(* CoDeSys 2.3.9.48 project: 5-hospital_Main_PLC.pro *)
(* Libraries: Standard.lib 20.5.14 09:13:26, Iecsfc.lib 30.1.13 14:05:12, SYSLIBCALLBACK.LIB 30.1.13 14:05:12, Modb_l05.lib 13.5.15 11:30:08, mod_com.lib 30.1.13 14:05:12, Serial_Interface_01.lib 22.4.13 13:50:14, SerComm.lib 30.1.13 14:05:12, Wago_MBCFG_SERIAL_01.lib 1.4.15 15:24:28, Wago_MBCFG_COMMON_01.lib 1.4.15 15:24:28 *)

(* PLC configuration (modules and I/O channels)
K-Bus [K_Bus] node 0, in %IB0 out %QB0 {KbusBusMode = 1; KbusCycleTime = 10000; KbusThreadPriority = 0; KbusSetOutputsToZeroOnApplicationStop = 1}
Modbus variables [PFC200MODBUS] node 1, in %IB0 out %QB0 {PlcStopBehaviour = 1; FiledbusErrorBehaviour = 1; TcpOperation = 1; TcpPort = 502; TcpTimeout = 600; UdpOperation = 1; UdpPort = 502; RtuOperation = 0; NodeId = 1; ResponseTimeout = 5000; Interface = 0; Baud = 115200; StopBits = 1; Parity = 1; FlowCtrl = 0; PhysInterface = 0}
Modbus-Master [MB_MASTER] node 2, in %IB0 out %QB0
*)

(* POU PLC_PRG, ST *)
PROGRAM PLC_PRG
VAR
END_VAR

END_PROGRAM

(* POU Generated Code/Serial/MBCFG/MBCFG_COM_OBJECTS, ST *)
PROGRAM MBCFG_COM_OBJECTS
VAR_INPUT

      MBCFG_MB_COM_0	:	MBCFG_COM_SER_OBJECT := (   ASCII_Mode      := FALSE,
                                                     COM_PORT        := 0,	 
                                                     COM_BAUDRATE    := BAUD_9600,
                                                     COM_PARITY      := PARITY_NO,
                                                     COM_STOPBITS    := STOPBITS_1,
                                                     COM_BYTESIZE    := BS_8,
                                                     COM_FLOW_CONTROL:= HALFDUPLEX,
                                                     TIME_OUT        := t#100ms
                                                 );



END_VAR
;
END_PROGRAM

(* POU Generated Code/Serial/MBCFG_ModbusSlave, ST *)
PROGRAM MBCFG_ModbusSlave (* generated by config one prg for each slave *)

VAR_INPUT

END_VAR

VAR_OUTPUT
           xNewVar       :    BOOL;       (**) 


    (*--- system variables (read only) -------------------------*)
    MBCFG_SlaveAddress  :   USINT := 1; (* valid range 1..247   *)
    MBCFG_TimeOut       :   TIME  := t#20ms;
    MBCFG_RequestDelay  :   TIME  := t#0ms; (* 0 means no delay *)
    MBCFG_Error         :   MBCFG_eERROR := MBCFG_START_UP;
	MBCFG_SERCOM_ERROR  : 	BYTE; (* generated by sercomm.lib -> see documentation of sercomm.lib *)
	MBCFG_LastJob       :   MBCFG_typCOM_JOB;
    (*----------------------------------------------------------*)
END_VAR

{library private}
VAR CONSTANT
    zz_VARIABLECOUNT    :   INT := 1;   (* number of variables  *)
    zz_JOBCOUNT         :   INT := 1;   (* number of jobs       *)
END_VAR
VAR

    (*=== VARIABLE LIST ===============================================================================*)
    zz_VariableList :   ARRAY[1..zz_VARIABLECOUNT] OF MBCFG_typVARIABLE :=
        (    DataType        := MBCFG_TYPE_BOOL,
        ByteOrder       := MBCFG_BYTE_ORDER_0,
        BitSize         := 1,
        ptVar           := 0,
        ReadJobIndex    := 1,
        ReadStartBitNo  := 0,
        WriteJobIndex   := 0,
        WriteStartBitNo := 0 )

                        ;
    (*=================================================================================================*)

    (*=== JOB LIST ====================================================================================*)
    zz_JobList      :   ARRAY[1..zz_JOBCOUNT] OF MBCFG_typCOM_JOB :=
         (   Functioncode            := 3,
        ReadStartAddress        := 1,
        ReadQuantity            := 1,
        WriteStartAddress       := 0,
        WriteQuantity           := 0,
        ptReadData              := 0, 
        ptWriteData             := 0 )

                        ;
    (*=================================================================================================*)

    (*### MODBUS MASTER ##### FIXED CODE ###########################################*)
    zz_MBCFG_MASTER			:	MBCFG_MASTER_SERIAL; (* for serial modbus RTU/ASCII *)
    (*##############################################################################*)

END_VAR
(*--- for each variable one entry ------------------------------------*)
   zz_VariableList[1].ptVar := ADR(xNewVar);

(*--------------------------------------------------------------------*)


(*=== call of the master for this slave ====================================================*)
zz_MBCFG_MASTER(   usiSlaveAddress  := MBCFG_SlaveAddress,               (* fixed entry     *)
                    tTimeOut        := MBCFG_TimeOut,                    (* fixed entry     *)
                    iVariableCount  := zz_VARIABLECOUNT,                 (* fixed entry     *)
                    ptVariableList  := ADR(zz_VariableList),             (* fixed entry     *)
                    iJobCount       := zz_JOBCOUNT,                      (* fixed entry     *)
                    ptJobList       := ADR(zz_JobList),                  (* fixed entry     *)
                    tRequestDelay   := MBCFG_RequestDelay,               (* fixed entry     *)
                    MB_ComObject    := MBCFG_COM_OBJECTS.MBCFG_MB_COM_0,(* generated entry *)
                    eError          => MBCFG_Error,                      (* fixed entry     *)
                    LastJob         => MBCFG_LastJob                     (* fixed entry     *)
                );
(*==========================================================================================*)

MBCFG_SERCOM_ERROR := MBCFG_COM_OBJECTS.MBCFG_MB_COM_0.bInterfaceError; 
END_PROGRAM

(* POU Generated Code/Serial/MBCFG_ModbusSlave0, ST *)
PROGRAM MBCFG_ModbusSlave0 (* generated by config one prg for each slave *)

VAR_INPUT
       xNewVar1       :    BOOL;       (**) 

END_VAR

VAR_OUTPUT
    

    (*--- system variables (read only) -------------------------*)
    MBCFG_SlaveAddress  :   USINT := 2; (* valid range 1..247   *)
    MBCFG_TimeOut       :   TIME  := t#20ms;
    MBCFG_RequestDelay  :   TIME  := t#0ms; (* 0 means no delay *)
    MBCFG_Error         :   MBCFG_eERROR := MBCFG_START_UP;
	MBCFG_SERCOM_ERROR  : 	BYTE; (* generated by sercomm.lib -> see documentation of sercomm.lib *)
	MBCFG_LastJob       :   MBCFG_typCOM_JOB;
    (*----------------------------------------------------------*)
END_VAR

{library private}
VAR CONSTANT
    zz_VARIABLECOUNT    :   INT := 1;   (* number of variables  *)
    zz_JOBCOUNT         :   INT := 1;   (* number of jobs       *)
END_VAR
VAR

    (*=== VARIABLE LIST ===============================================================================*)
    zz_VariableList :   ARRAY[1..zz_VARIABLECOUNT] OF MBCFG_typVARIABLE :=
        (    DataType        := MBCFG_TYPE_BOOL,
        ByteOrder       := MBCFG_BYTE_ORDER_0,
        BitSize         := 1,
        ptVar           := 0,
        ReadJobIndex    := 0,
        ReadStartBitNo  := 0,
        WriteJobIndex   := 1,
        WriteStartBitNo := 0 )

                        ;
    (*=================================================================================================*)

    (*=== JOB LIST ====================================================================================*)
    zz_JobList      :   ARRAY[1..zz_JOBCOUNT] OF MBCFG_typCOM_JOB :=
         (   Functioncode            := 5,
        ReadStartAddress        := 0,
        ReadQuantity            := 0,
        WriteStartAddress       := 0,
        WriteQuantity           := 1,
        ptReadData              := 0, 
        ptWriteData             := 0 )

                        ;
    (*=================================================================================================*)

    (*### MODBUS MASTER ##### FIXED CODE ###########################################*)
    zz_MBCFG_MASTER			:	MBCFG_MASTER_SERIAL; (* for serial modbus RTU/ASCII *)
    (*##############################################################################*)

END_VAR
(*--- for each variable one entry ------------------------------------*)
   zz_VariableList[1].ptVar := ADR(xNewVar1);

(*--------------------------------------------------------------------*)


(*=== call of the master for this slave ====================================================*)
zz_MBCFG_MASTER(   usiSlaveAddress  := MBCFG_SlaveAddress,               (* fixed entry     *)
                    tTimeOut        := MBCFG_TimeOut,                    (* fixed entry     *)
                    iVariableCount  := zz_VARIABLECOUNT,                 (* fixed entry     *)
                    ptVariableList  := ADR(zz_VariableList),             (* fixed entry     *)
                    iJobCount       := zz_JOBCOUNT,                      (* fixed entry     *)
                    ptJobList       := ADR(zz_JobList),                  (* fixed entry     *)
                    tRequestDelay   := MBCFG_RequestDelay,               (* fixed entry     *)
                    MB_ComObject    := MBCFG_COM_OBJECTS.MBCFG_MB_COM_0,(* generated entry *)
                    eError          => MBCFG_Error,                      (* fixed entry     *)
                    LastJob         => MBCFG_LastJob                     (* fixed entry     *)
                );
(*==========================================================================================*)

MBCFG_SERCOM_ERROR := MBCFG_COM_OBJECTS.MBCFG_MB_COM_0.bInterfaceError; 
END_PROGRAM

(* POU Configuration/MODBUS_CONFIGURATION, ST *)
PROGRAM MODBUS_CONFIGURATION        
VAR                                
END_VAR                            
(*                                 
   <?xml version="1.0" encoding="UTF-16" standalone="yes"?>
<network xml_structure_version="1" xml_feature_version="1">
	<generator_settings minRTUTaskCycleTimeMs="5" minEthaskCycleTimeMs="5" ethSlaveMultiplier="0.1" rtuInterfaceMultiplier="0.1" taskGeneration="true"/>
	<master_interface type="serial" name="Configuration Root Node" com_port="0" baudrate="9600" databits="8" stopbits="1" parity="no" hwtype="RS485" flow_control="Xon/Xoff" asciimode="false" expanded="true">
		<mb_slave comment="" name="ModbusSlave" expanded="true" type="generic">
			<mb_connection type="serial" unitid="1" request_delay_ms="0" response_timeout_ms="20"/>
			<generic_vars comment="" expanded="true">
				<generic_var data_type="BOOL">
					<generic_params name="xNewVar" comment="" expanded="false" mb_iotype="unused" mb_access="ro" var_byteorder="B1B2B3B4"/>
					<mb_address explicitAccess="false" FCRead="3" FCWrite="0" ReadMBAddress="1" WriteMBAddress="0" ReadBitOffset="0" WriteBitOffset="0"/>
				</generic_var>
			</generic_vars>
		</mb_slave>
		<mb_slave comment="" name="ModbusSlave0" expanded="true" type="generic">
			<mb_connection type="serial" unitid="2" request_delay_ms="0" response_timeout_ms="20"/>
			<generic_vars comment="" expanded="true">
				<generic_var data_type="BOOL">
					<generic_params name="xNewVar1" comment="" expanded="true" mb_iotype="unused" mb_access="wo" var_byteorder="B1B2B3B4"/>
					<mb_address explicitAccess="false" FCRead="0" FCWrite="5" ReadMBAddress="0" WriteMBAddress="0" ReadBitOffset="0" WriteBitOffset="0"/>
				</generic_var>
			</generic_vars>
		</mb_slave>
	</master_interface>
</network>
                              
*)                                 
;                                  
END_PROGRAM
